INTERFACE I_Light

PROPERTY bIsOn : BOOL
GET
END_GET
END_PROPERTY

METHOD changeBrightness : BOOL
VAR_INPUT
	in_rNewBrightness	:REAL;
END_VAR
END_METHOD

METHOD changeColor : BOOL
VAR_INPUT
	in_eNewColor	:E_ColorCodes;
END_VAR
END_METHOD

PROPERTY eColor : E_ColorCodes
GET
END_GET
END_PROPERTY

PROPERTY rBrightness : REAL
GET
END_GET
END_PROPERTY

METHOD turnLightOff : BOOL
VAR_INPUT
END_VAR
END_METHOD

METHOD turnLightOn : BOOL
VAR_INPUT
END_VAR
END_METHOD

END_INTERFACE

(* stored: Version 1.1.0.1
   Itf I_Light: Id {8ad8afa3-1d92-4135-8ad6-42218d8d7506}
   Property bIsOn: Id {f80d03a0-8d7f-4fbd-b11f-fdf07e6907ec}
   Get Get: Id {38267145-8e9e-4060-bb49-626265b16652}
   Method changeBrightness: Id {e349acd3-ff6c-4876-8841-3ca034b8cb63}
   Method changeColor: Id {fe63f06c-5c3b-4a8c-b3aa-661684998043}
   Property eColor: Id {95abfeba-0e79-41a2-a8b1-ce6458a56102}
   Get Get: Id {4f2cbe78-ab39-48f7-ac28-c537038da46b}
   Property rBrightness: Id {53f67a20-62b6-4370-97a9-2d7b9abaffd6}
   Get Get: Id {a29d5c33-4824-46e5-aeb1-a0cfc5a2cd91}
   Method turnLightOff: Id {b61d4950-f124-48cb-88b4-8e2eadd227a1}
   Method turnLightOn: Id {e93f2052-179f-42e7-87f8-f4b96779fa36} *)
